// TIA Portal V17 export
// export: Created 2024-09-03T21:55:01.0772664Z, ExportSetting WithDefaults, DisplayName Totally Integrated Automation Portal, DisplayVersion V17 Update 7, DisplayName TIA Portal Openness, DisplayVersion V17 Update 7, DisplayName TIA Portal Version Control Interface, DisplayVersion V17, DisplayName SINAMICS Startdrive Advanced, DisplayVersion V17 SP2, DisplayName SINAMICS Startdrive G110M, G120, G120C, G120D, G120P, G115D, DisplayVersion V17 SP2, DisplayName SINAMICS Startdrive G130, G150, S120, S150, SINAMICS MV, S210, DisplayVersion V17 SP2, DisplayName STEP 7 Professional, DisplayVersion V17 Update 7, DisplayName STEP 7 Safety, DisplayVersion V17 Update 6, DisplayName WinCC Advanced / Unified PC, DisplayVersion V17 Update 7
FUNCTION "DATOS_IJCORE" : Void   // FC1, LAD
{ S7_Optimized_Access := 'TRUE' }
VERSION : 0.1
// stored: AutoNumber true, IsIECCheckEnabled false, SetENOAutomatically false, UDAEnableTagReadback false
   VAR_TEMP
      ijc_off : Bool;
      PV_HMI : Int;
      INDEX_HMI2 : Int;
      INDEX_HMI3 : Int;
   END_VAR
   VAR_TEMP   // added for the SCL form of the ladder/FBD networks
      _w1 : Bool;
   END_VAR
BEGIN

REGION Network 2: ALARMA ACTIVA
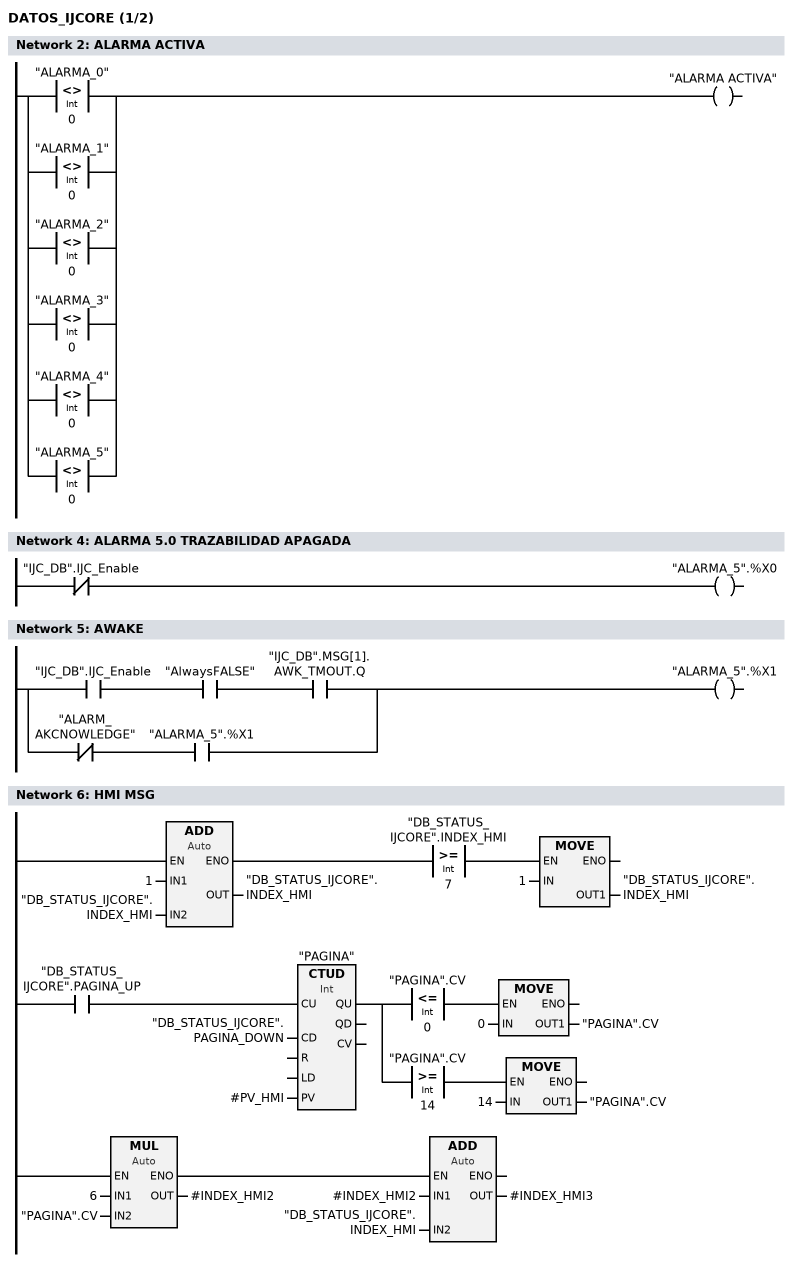
   RUNG wire#powerrail
      { S7_Templates := "SrcType := Int" } NE_Contact(in1 := "ALARMA_0", in2 := 0)
      wire#w1
      Coil( "ALARMA ACTIVA" )
   END_RUNG
   RUNG wire#powerrail
      { S7_Templates := "SrcType := Int" } NE_Contact(in1 := "ALARMA_1", in2 := 0)
   END_RUNG wire#w1
   RUNG wire#powerrail
      { S7_Templates := "SrcType := Int" } NE_Contact(in1 := "ALARMA_2", in2 := 0)
   END_RUNG wire#w1
   RUNG wire#powerrail
      { S7_Templates := "SrcType := Int" } NE_Contact(in1 := "ALARMA_3", in2 := 0)
   END_RUNG wire#w1
   RUNG wire#powerrail
      { S7_Templates := "SrcType := Int" } NE_Contact(in1 := "ALARMA_4", in2 := 0)
   END_RUNG wire#w1
   RUNG wire#powerrail
      { S7_Templates := "SrcType := Int" } NE_Contact(in1 := "ALARMA_5", in2 := 0)
   END_RUNG wire#w1
   // the same network as SCL:
   "ALARMA ACTIVA" := ("ALARMA_0" <> 0) OR ("ALARMA_1" <> 0) OR ("ALARMA_2" <> 0) OR ("ALARMA_3" <> 0) OR ("ALARMA_4" <> 0) OR ("ALARMA_5" <> 0);
END_REGION

REGION Network 3 (SCL): ALARMAS IJCORE

   //////// MESAGE ALARMS /////////
   //
   //Alarm AWAKE  error
   //
   IF "IJC_DB".AWAKE_SIGNAL_INSTANCE.AwSignalTimeOutFault AND"IJC_DB".IJC_Enable THEN
       "Alarms".Alarm[127] := true;
   ELSE
       "Alarms".Alarm[127] := FALSE;
   END_IF;

   CASE "DB_ProductionProgramActual".Program.MechanicalType OF
       1:

           //Alarm IJC STA SIDE MEMBER LH  error
           //
           IF "IJC_DB".MSG[1].DN AND "DB_STATUS_IJCORE".ANSWER_STA[1] = -2
               AND "IJC_DB".IJC_Enable AND "DB_ProductionProgramActual".Program.MechanicalType = 1 THEN
               "Alarms".Alarm[130] := true;
           ELSE
               "Alarms".Alarm[130] := FALSE;
           END_IF;

           IF "IJC_DB".MSG[1].DN AND "DB_STATUS_IJCORE".ANSWER_STA[1] = -10
               AND "IJC_DB".IJC_Enable AND "DB_ProductionProgramActual".Program.MechanicalType = 1 THEN
               "Alarms".Alarm[150] := true;
           ELSE
               "Alarms".Alarm[150] := FALSE;
           END_IF;

           IF "IJC_DB".MSG[1].DN AND "DB_STATUS_IJCORE".ANSWER_STA[1] = -16
               AND "IJC_DB".IJC_Enable AND "DB_ProductionProgramActual".Program.MechanicalType = 1 THEN
               "Alarms".Alarm[151] := true;
           ELSE
               "Alarms".Alarm[151] := FALSE;
           END_IF;

           IF "IJC_DB".MSG[1].DN AND "DB_STATUS_IJCORE".ANSWER_STA[1] = 8224
               AND "IJC_DB".IJC_Enable AND "DB_ProductionProgramActual".Program.MechanicalType = 1 THEN
               "Alarms".Alarm[152] := true;
           ELSE
               "Alarms".Alarm[152] := FALSE;
           END_IF;

           //Alarm IJC STA SIDE MEMBER RH  error
           //
           IF "IJC_DB".MSG[2].DN AND "DB_STATUS_IJCORE".ANSWER_STA[2] = -2
               AND "IJC_DB".IJC_Enable THEN
               "Alarms".Alarm[131] := true;
           ELSE
               "Alarms".Alarm[131] := FALSE;
           END_IF;

           IF "IJC_DB".MSG[2].DN AND "DB_STATUS_IJCORE".ANSWER_STA[2] = -10
               AND "IJC_DB".IJC_Enable THEN
               "Alarms".Alarm[153] := true;
           ELSE
               "Alarms".Alarm[153] := FALSE;
           END_IF;

           IF "IJC_DB".MSG[2].DN AND "DB_STATUS_IJCORE".ANSWER_STA[2] = -16
               AND "IJC_DB".IJC_Enable THEN
               "Alarms".Alarm[154] := true;
           ELSE
               "Alarms".Alarm[154] := FALSE;
           END_IF;

           IF "IJC_DB".MSG[2].DN AND "DB_STATUS_IJCORE".ANSWER_STA[2] = 8224
               AND "IJC_DB".IJC_Enable THEN
               "Alarms".Alarm[155] := true;
           ELSE
               "Alarms".Alarm[155] := FALSE;
           END_IF;
       0:

           //Alarm IJC STA SIDE MEMBER LH  error
           //
           IF "IJC_DB".MSG[1].DN AND "DB_STATUS_IJCORE".ANSWER_STA[1] = -2
               AND "IJC_DB".IJC_Enable AND "DB_ProductionProgramActual".Program.MechanicalType = 1 THEN
               "Alarms".Alarm[131] := true;
           ELSE
               "Alarms".Alarm[131] := FALSE;
           END_IF;

           IF "IJC_DB".MSG[1].DN AND "DB_STATUS_IJCORE".ANSWER_STA[1] = -10
               AND "IJC_DB".IJC_Enable AND "DB_ProductionProgramActual".Program.MechanicalType = 1 THEN
               "Alarms".Alarm[153] := true;
           ELSE
               "Alarms".Alarm[153] := FALSE;
           END_IF;

           IF "IJC_DB".MSG[1].DN AND "DB_STATUS_IJCORE".ANSWER_STA[1] = -16
               AND "IJC_DB".IJC_Enable AND "DB_ProductionProgramActual".Program.MechanicalType = 1 THEN
               "Alarms".Alarm[154] := true;
           ELSE
               "Alarms".Alarm[154] := FALSE;
           END_IF;

           IF "IJC_DB".MSG[1].DN AND "DB_STATUS_IJCORE".ANSWER_STA[1] = 8224
               AND "IJC_DB".IJC_Enable AND "DB_ProductionProgramActual".Program.MechanicalType = 1 THEN
               "Alarms".Alarm[155] := true;
           ELSE
               "Alarms".Alarm[155] := FALSE;
           END_IF;

           //Alarm IJC STA SIDE MEMBER RH  error
           //
           IF "IJC_DB".MSG[2].DN AND "DB_STATUS_IJCORE".ANSWER_STA[2] = -2
               AND "IJC_DB".IJC_Enable THEN
               "Alarms".Alarm[130] := true;
           ELSE
               "Alarms".Alarm[130] := FALSE;
           END_IF;

           IF "IJC_DB".MSG[2].DN AND "DB_STATUS_IJCORE".ANSWER_STA[2] = -10
               AND "IJC_DB".IJC_Enable THEN
               "Alarms".Alarm[150] := true;
           ELSE
               "Alarms".Alarm[150] := FALSE;
           END_IF;

           IF "IJC_DB".MSG[2].DN AND "DB_STATUS_IJCORE".ANSWER_STA[2] = -16
               AND "IJC_DB".IJC_Enable THEN
               "Alarms".Alarm[151] := true;
           ELSE
               "Alarms".Alarm[151] := FALSE;
           END_IF;

           IF "IJC_DB".MSG[2].DN AND "DB_STATUS_IJCORE".ANSWER_STA[2] = 8224
               AND "IJC_DB".IJC_Enable THEN
               "Alarms".Alarm[152] := true;
           ELSE
               "Alarms".Alarm[152] := FALSE;
           END_IF;
   END_CASE;

   //Alarm IJC STA FRONT TUBE  error
   //
   IF "IJC_DB".MSG[3].DN AND "DB_STATUS_IJCORE".ANSWER_STA[3] = -2
       AND "IJC_DB".IJC_Enable THEN
       "Alarms".Alarm[132] := true;
   ELSE
       "Alarms".Alarm[132] := FALSE;
   END_IF;

   IF "IJC_DB".MSG[3].DN AND "DB_STATUS_IJCORE".ANSWER_STA[3] = -10
       AND "IJC_DB".IJC_Enable THEN
       "Alarms".Alarm[156] := true;
   ELSE
       "Alarms".Alarm[156] := FALSE;
   END_IF;

   IF "IJC_DB".MSG[3].DN AND "DB_STATUS_IJCORE".ANSWER_STA[3] = -16
       AND "IJC_DB".IJC_Enable THEN
       "Alarms".Alarm[157] := true;
   ELSE
       "Alarms".Alarm[157] := FALSE;
   END_IF;

   IF "IJC_DB".MSG[3].DN AND "DB_STATUS_IJCORE".ANSWER_STA[3] = 8224
       AND "IJC_DB".IJC_Enable THEN
       "Alarms".Alarm[158] := true;
   ELSE
       "Alarms".Alarm[158] := FALSE;
   END_IF;
   //Alarm IJC STA REAR TUBE  error
   //
   IF "IJC_DB".MSG[4].DN AND "DB_STATUS_IJCORE".ANSWER_STA[4] = -2
       AND "IJC_DB".IJC_Enable THEN
       "Alarms".Alarm[133] := true;
   ELSE
       "Alarms".Alarm[133] := FALSE;
   END_IF;

   IF "IJC_DB".MSG[4].DN AND "DB_STATUS_IJCORE".ANSWER_STA[4] = -10
       AND "IJC_DB".IJC_Enable THEN
       "Alarms".Alarm[159] := true;
   ELSE
       "Alarms".Alarm[159] := FALSE;
   END_IF;

   IF "IJC_DB".MSG[4].DN AND "DB_STATUS_IJCORE".ANSWER_STA[4] = -16
       AND "IJC_DB".IJC_Enable THEN
       "Alarms".Alarm[160] := true;
   ELSE
       "Alarms".Alarm[160] := FALSE;
   END_IF;

   IF "IJC_DB".MSG[4].DN AND "DB_STATUS_IJCORE".ANSWER_STA[4] = 8224
       AND "IJC_DB".IJC_Enable THEN
       "Alarms".Alarm[161] := true;
   ELSE
       "Alarms".Alarm[161] := FALSE;
   END_IF;

   //Alarm IJC TRC SIDE MEMBER LH  error
   //
   IF "IJC_DB".MSG[5].DN AND "DB_STATUS_IJCORE".ANSWER_TRC[1] = -2
       AND "IJC_DB".IJC_Enable AND NOT "M_TRC1_OK" THEN
       "Alarms".Alarm[134] := true;
   ELSE
       "Alarms".Alarm[134] := FALSE;
   END_IF;

   IF "IJC_DB".MSG[5].DN AND "DB_STATUS_IJCORE".ANSWER_TRC[1] = -4
       AND "IJC_DB".IJC_Enable AND NOT "M_TRC1_OK" THEN
       "Alarms".Alarm[162] := true;
   ELSE
       "Alarms".Alarm[162] := FALSE;
   END_IF;

   IF "IJC_DB".MSG[5].DN AND "DB_STATUS_IJCORE".ANSWER_TRC[1] = -16
       AND "IJC_DB".IJC_Enable AND NOT "M_TRC1_OK" THEN
       "Alarms".Alarm[163] := true;
   ELSE
       "Alarms".Alarm[163] := FALSE;
   END_IF;

   IF "IJC_DB".MSG[5].DN AND "DB_STATUS_IJCORE".ANSWER_TRC[1] = 8224
       AND "IJC_DB".IJC_Enable AND NOT "M_TRC1_OK" THEN
       "Alarms".Alarm[146] := true;
   ELSE
       "Alarms".Alarm[146] := FALSE;
   END_IF;

   //Alarm IJC TRC SIDE MEMBER RH  error
   //
   IF "IJC_DB".MSG[6].DN AND "DB_STATUS_IJCORE".ANSWER_TRC[2] = -2
       AND "IJC_DB".IJC_Enable AND NOT "M_TRC2_OK" THEN
       "Alarms".Alarm[135] := true;
   ELSE
       "Alarms".Alarm[135] := FALSE;
   END_IF;

   IF "IJC_DB".MSG[6].DN AND "DB_STATUS_IJCORE".ANSWER_TRC[2] = -4
       AND "IJC_DB".IJC_Enable AND NOT "M_TRC2_OK" THEN
       "Alarms".Alarm[164] := true;
   ELSE
       "Alarms".Alarm[164] := FALSE;
   END_IF;

   IF "IJC_DB".MSG[6].DN AND "DB_STATUS_IJCORE".ANSWER_TRC[2] = -16
       AND "IJC_DB".IJC_Enable AND NOT "M_TRC2_OK" THEN
       "Alarms".Alarm[165] := true;
   ELSE
       "Alarms".Alarm[165] := FALSE;
   END_IF;

   IF "IJC_DB".MSG[6].DN AND "DB_STATUS_IJCORE".ANSWER_TRC[2] = 8224
       AND "IJC_DB".IJC_Enable AND NOT "M_TRC2_OK" THEN
       "Alarms".Alarm[147] := true;
   ELSE
       "Alarms".Alarm[147] := FALSE;
   END_IF;

   //Alarm IJC TRC FRONT TUBE  error
   //
   IF "IJC_DB".MSG[7].DN AND "DB_STATUS_IJCORE".ANSWER_TRC[3] = -2
       AND "IJC_DB".IJC_Enable AND NOT "M_TRC3_OK" THEN
       "Alarms".Alarm[136] := true;
   ELSE
       "Alarms".Alarm[136] := FALSE;
   END_IF;

   IF "IJC_DB".MSG[7].DN AND "DB_STATUS_IJCORE".ANSWER_TRC[3] = -4
       AND "IJC_DB".IJC_Enable AND NOT "M_TRC3_OK" THEN
       "Alarms".Alarm[166] := true;
   ELSE
       "Alarms".Alarm[166] := FALSE;
   END_IF;

   IF "IJC_DB".MSG[7].DN AND "DB_STATUS_IJCORE".ANSWER_TRC[3] = -16
       AND "IJC_DB".IJC_Enable AND NOT "M_TRC3_OK" THEN
       "Alarms".Alarm[167] := true;
   ELSE
       "Alarms".Alarm[167] := FALSE;
   END_IF;

   IF "IJC_DB".MSG[7].DN AND "DB_STATUS_IJCORE".ANSWER_TRC[3] = 8224
       AND "IJC_DB".IJC_Enable AND NOT "M_TRC3_OK" THEN
       "Alarms".Alarm[148] := true;
   ELSE
       "Alarms".Alarm[148] := FALSE;
   END_IF;
   //Alarm IJC TRC REAR TUBE  error
   //
   IF "IJC_DB".MSG[8].DN AND "DB_STATUS_IJCORE".ANSWER_TRC[4] = -2
       AND "IJC_DB".IJC_Enable AND NOT "M_TRC4_OK" THEN
       "Alarms".Alarm[137] := true;
   ELSE
       "Alarms".Alarm[137] := FALSE;
   END_IF;

   IF "IJC_DB".MSG[8].DN AND "DB_STATUS_IJCORE".ANSWER_TRC[4] = -4
       AND "IJC_DB".IJC_Enable AND NOT "M_TRC4_OK" THEN
       "Alarms".Alarm[168] := true;
   ELSE
       "Alarms".Alarm[168] := FALSE;
   END_IF;

   IF "IJC_DB".MSG[8].DN AND "DB_STATUS_IJCORE".ANSWER_TRC[4] = -16
       AND "IJC_DB".IJC_Enable AND NOT "M_TRC4_OK" THEN
       "Alarms".Alarm[169] := true;
   ELSE
       "Alarms".Alarm[169] := FALSE;
   END_IF;

   IF "IJC_DB".MSG[8].DN AND "DB_STATUS_IJCORE".ANSWER_TRC[4] <> 8224
       AND "IJC_DB".IJC_Enable AND NOT "M_TRC4_OK" THEN
       "Alarms".Alarm[149] := true;
   ELSE
       "Alarms".Alarm[149] := FALSE;
   END_IF;
   //Alarm IJC TRR 1 CUPFORMIG error
   //
   //IF "IJC_DB".MSG[9].DN AND "DB_STATUS_IJCORE".ANSWER_RECIB[9] = -2
      // AND "IJC_DB".IJC_Enable THEN
       //"Alarms".Alarm[122] := true;
   //ELSE
     //  "Alarms".Alarm[122] := FALSE;
   //END_IF;
   //
   ////IF "IJC_DB".MSG[9].DN AND "DB_STATUS_IJCORE".ANSWER_RECIB[9] = -16
   // AND "IJC_DB".IJC_Enable THEN
   //"Alarms".Alarm[122] := true;
   //ELSE
   //  "Alarms".Alarm[122] := FALSE;
   //END_IF;
   //
   //IF "IJC_DB".MSG[9].DN AND "DB_STATUS_IJCORE".ANSWER_RECIB[9] = 8224
   // AND "IJC_DB".IJC_Enable THEN
   //"Alarms".Alarm[122] := true;
   //ELSE
   //  "Alarms".Alarm[122] := FALSE;
   //END_IF;

   //Alarm IJC TRR 2 RIVETS error
   //
   //IF "IJC_DB".MSG[10].DN AND "DB_STATUS_IJCORE".ANSWER_RECIB[10] = -2
       //AND "IJC_DB".IJC_Enable THEN
       //"Alarms".Alarm[123] := true;
   //ELSE
     //  "Alarms".Alarm[123] := FALSE;
   //END_IF;
   //
   //IF "IJC_DB".MSG[10].DN AND "DB_STATUS_IJCORE".ANSWER_RECIB[10] = -16
   //AND "IJC_DB".IJC_Enable THEN
   //"Alarms".Alarm[123] := true;
   //ELSE
   //  "Alarms".Alarm[123] := FALSE;
   //END_IF;
   //
   //IF "IJC_DB".MSG[10].DN AND "DB_STATUS_IJCORE".ANSWER_RECIB[10] = 8224
   //AND "IJC_DB".IJC_Enable THEN
   //"Alarms".Alarm[123] := true;
   //ELSE
   //  "Alarms".Alarm[123] := FALSE;
   //END_IF;

   //Alarm IJC CNF SIDE MEMBER LH  error
   //
   //IF "IJC_DB".MSG[11].DN AND "DB_STATUS_IJCORE".ANSWER_RECIB[11] <> 1
     //  AND "IJC_DB".IJC_Enable THEN
     //  "Alarms".Alarm[124] := true;
   //END_IF;
   //

   //
   //IF "IJC_DB".MSG[11].DN AND "DB_STATUS_IJCORE".ANSWER_RECIB[11] = 8224
   //  AND "IJC_DB".IJC_Enable THEN
   //  "Alarms".Alarm[124] := true;
   //END_IF;

   //Alarm IJC CNF SIDE MEMBER RH  error
   //
   //IF "IJC_DB".MSG[12].DN AND "DB_STATUS_IJCORE".ANSWER_RECIB[12] <> 1
     //  AND "IJC_DB".IJC_Enable THEN
       //"Alarms".Alarm[124] := true;
   //END_IF;

   //Alarm IJC CNF REAR TUBE  error
   //
   //IF "IJC_DB".MSG[13].DN AND "DB_STATUS_IJCORE".ANSWER_RECIB[13] <> 1
     //  AND "IJC_DB".IJC_Enable THEN
       //"Alarms".Alarm[125] := true;
   //ELSE
     //  "Alarms".Alarm[125] := FALSE;
   //END_IF;

   //Alarm IJC CNF SIDE MEMBER LH  error
   //
   //IF "IJC_DB".MSG[15].DN AND "DB_STATUS_IJCORE".ANSWER_RECIB[15] <> 1
     //  AND "IJC_DB".IJC_Enable THEN
       //"Alarms".Alarm[126] := true;
   //ELSE
     //  "Alarms".Alarm[126] := FALSE;
   //END_IF;
   //
   //Alarm IJC PFC SIDE MEMBER LH  error
   //
   IF "IJC_DB".MSG[14].DN AND "DB_STATUS_IJCORE".ANSWER_RECIB[14] = -2
       AND "IJC_DB".IJC_Enable AND NOT "M_PFC_OK" THEN
       "Alarms".Alarm[170] := true;
   ELSE
       "Alarms".Alarm[170] := FALSE;
   END_IF;

   IF "IJC_DB".MSG[14].DN AND "DB_STATUS_IJCORE".ANSWER_RECIB[14] = -4
       AND "IJC_DB".IJC_Enable AND NOT "M_PFC_OK" THEN
       "Alarms".Alarm[143] := true;
   ELSE
       "Alarms".Alarm[143] := FALSE;
   END_IF;

   IF "IJC_DB".MSG[14].DN AND "DB_STATUS_IJCORE".ANSWER_RECIB[14] = -10
       AND "IJC_DB".IJC_Enable AND NOT "M_PFC_OK" THEN
      "Alarms".Alarm[171] := true;
   ELSE
     "Alarms".Alarm[171] := FALSE;
   END_IF;


   IF "IJC_DB".MSG[14].DN AND "DB_STATUS_IJCORE".ANSWER_RECIB[14] = -16
       AND "IJC_DB".IJC_Enable AND NOT "M_PFC_OK" THEN
     "Alarms".Alarm[172] := true;
   ELSE
       "Alarms".Alarm[172] := FALSE;
   END_IF;

   IF "IJC_DB".MSG[14].DN AND "DB_STATUS_IJCORE".ANSWER_RECIB[14] = 8224
       AND "IJC_DB".IJC_Enable AND NOT "M_PFC_OK" THEN
       "Alarms".Alarm[145] := true;
   ELSE
       "Alarms".Alarm[145] := FALSE;
   END_IF;
END_REGION

REGION Network 4: ALARMA 5.0 TRAZABILIDAD APAGADA
   RUNG wire#powerrail
      I_Contact( "IJC_DB".IJC_Enable )
      Coil( "ALARMA_5".%X0 )
   END_RUNG
   // the same network as SCL:
   "ALARMA_5".%X0 := NOT "IJC_DB".IJC_Enable;
END_REGION

REGION Network 5: AWAKE
   RUNG wire#powerrail
      Contact( "IJC_DB".IJC_Enable )
      Contact( "AlwaysFALSE" )
      Contact( "IJC_DB".MSG[1].AWK_TMOUT.Q )
      wire#w1
      Coil( "ALARMA_5".%X1 )
   END_RUNG
   RUNG wire#powerrail
      I_Contact( "ALARM_AKCNOWLEDGE" )
      Contact( "ALARMA_5".%X1 )
   END_RUNG wire#w1
   // the same network as SCL:
   "ALARMA_5".%X1 := ("IJC_DB".IJC_Enable AND "AlwaysFALSE" AND "IJC_DB".MSG[1].AWK_TMOUT.Q) OR (NOT "ALARM_AKCNOWLEDGE" AND "ALARMA_5".%X1);
END_REGION

REGION Network 6: HMI MSG
   RUNG wire#powerrail
      Add(in1 := 1, in2 := "DB_STATUS_IJCORE".INDEX_HMI, out => "DB_STATUS_IJCORE".INDEX_HMI)
      { S7_Templates := "SrcType := Int" } GE_Contact(in1 := "DB_STATUS_IJCORE".INDEX_HMI, in2 := 7)
      Move(in := 1, out1 => "DB_STATUS_IJCORE".INDEX_HMI)
   END_RUNG
   RUNG wire#powerrail
      Contact( "DB_STATUS_IJCORE".PAGINA_UP )
      { S7_Templates := "value_type := Int" } "PAGINA".CTUD(cd := "DB_STATUS_IJCORE".PAGINA_DOWN, r :=, ld :=, pv := #PV_HMI, qd =>, cv =>)
      wire#w1
      { S7_Templates := "SrcType := Int" } LE_Contact(in1 := "PAGINA".CV, in2 := 0)
      Move(in := 0, out1 => "PAGINA".CV)
   END_RUNG
   RUNG wire#w1
      { S7_Templates := "SrcType := Int" } GE_Contact(in1 := "PAGINA".CV, in2 := 14)
      Move(in := 14, out1 => "PAGINA".CV)
   END_RUNG
   RUNG wire#powerrail
      Mul(in1 := 6, in2 := "PAGINA".CV, out => #INDEX_HMI2)
      Add(in1 := #INDEX_HMI2, in2 := "DB_STATUS_IJCORE".INDEX_HMI, out => #INDEX_HMI3)
   END_RUNG
   // the same network as SCL:
   "DB_STATUS_IJCORE".INDEX_HMI := 1 + "DB_STATUS_IJCORE".INDEX_HMI;
   IF "DB_STATUS_IJCORE".INDEX_HMI >= 7 THEN "DB_STATUS_IJCORE".INDEX_HMI := 1; END_IF;
   "PAGINA".CTUD(CU := "DB_STATUS_IJCORE".PAGINA_UP, CD := "DB_STATUS_IJCORE".PAGINA_DOWN, PV := #PV_HMI);
   #_w1 := "PAGINA".QU;
   IF "PAGINA".QU AND ("PAGINA".CV <= 0) THEN "PAGINA".CV := 0; END_IF;
   IF #_w1 AND ("PAGINA".CV >= 14) THEN "PAGINA".CV := 14; END_IF;
   #INDEX_HMI2 := 6 * "PAGINA".CV;
   #INDEX_HMI3 := #INDEX_HMI2 + "DB_STATUS_IJCORE".INDEX_HMI;
END_REGION

REGION Network 7: VARIABLES HMI
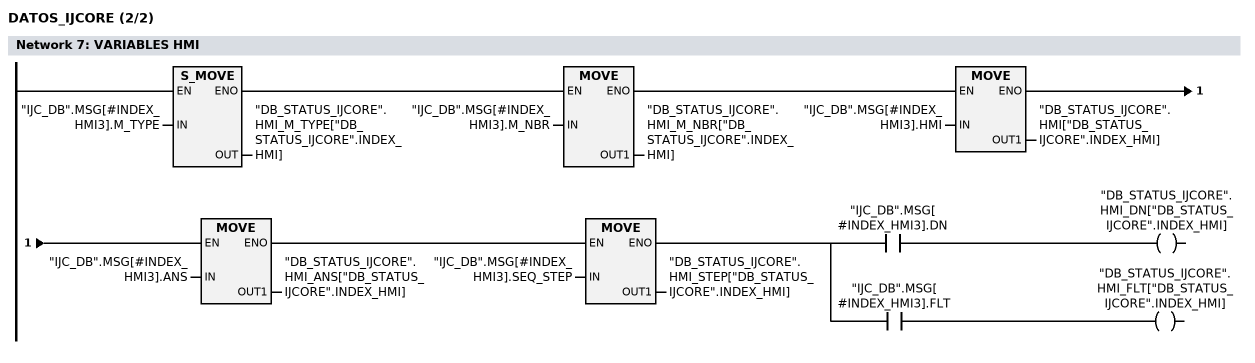
   RUNG wire#powerrail
      S_Move(in := "IJC_DB".MSG[#INDEX_HMI3].M_TYPE, out => "DB_STATUS_IJCORE".HMI_M_TYPE["DB_STATUS_IJCORE".INDEX_HMI])
      Move(in := "IJC_DB".MSG[#INDEX_HMI3].M_NBR, out1 => "DB_STATUS_IJCORE".HMI_M_NBR["DB_STATUS_IJCORE".INDEX_HMI])
      Move(in := "IJC_DB".MSG[#INDEX_HMI3].HMI, out1 => "DB_STATUS_IJCORE".HMI["DB_STATUS_IJCORE".INDEX_HMI])
      Move(in := "IJC_DB".MSG[#INDEX_HMI3].ANS, out1 => "DB_STATUS_IJCORE".HMI_ANS["DB_STATUS_IJCORE".INDEX_HMI])
      Move(in := "IJC_DB".MSG[#INDEX_HMI3].SEQ_STEP, out1 => "DB_STATUS_IJCORE".HMI_STEP["DB_STATUS_IJCORE".INDEX_HMI])
      wire#w1
      Contact( "IJC_DB".MSG[#INDEX_HMI3].DN )
      Coil( "DB_STATUS_IJCORE".HMI_DN["DB_STATUS_IJCORE".INDEX_HMI] )
   END_RUNG
   RUNG wire#w1
      Contact( "IJC_DB".MSG[#INDEX_HMI3].FLT )
      Coil( "DB_STATUS_IJCORE".HMI_FLT["DB_STATUS_IJCORE".INDEX_HMI] )
   END_RUNG
   // the same network as SCL:
   "DB_STATUS_IJCORE".HMI_M_TYPE["DB_STATUS_IJCORE".INDEX_HMI] := "IJC_DB".MSG[#INDEX_HMI3].M_TYPE;
   "DB_STATUS_IJCORE".HMI_M_NBR["DB_STATUS_IJCORE".INDEX_HMI] := "IJC_DB".MSG[#INDEX_HMI3].M_NBR;
   "DB_STATUS_IJCORE".HMI["DB_STATUS_IJCORE".INDEX_HMI] := "IJC_DB".MSG[#INDEX_HMI3].HMI;
   "DB_STATUS_IJCORE".HMI_ANS["DB_STATUS_IJCORE".INDEX_HMI] := "IJC_DB".MSG[#INDEX_HMI3].ANS;
   "DB_STATUS_IJCORE".HMI_STEP["DB_STATUS_IJCORE".INDEX_HMI] := "IJC_DB".MSG[#INDEX_HMI3].SEQ_STEP;
   "DB_STATUS_IJCORE".HMI_DN["DB_STATUS_IJCORE".INDEX_HMI] := "IJC_DB".MSG[#INDEX_HMI3].DN;
   "DB_STATUS_IJCORE".HMI_FLT["DB_STATUS_IJCORE".INDEX_HMI] := "IJC_DB".MSG[#INDEX_HMI3].FLT;
END_REGION
END_FUNCTION
